// TIA Portal project "babu_mathQuestions" (V15)

(* hardware
DEVICE "S7-1200 station_1"  S7-1200 Station
   slot 0: "Rack_0"  S7-1200 Rack  Rack  V1.0
   slot 1: "PLC_1"  CPU 1212C DC/DC/DC  6ES7 212-1AE40-0XB0  V4.2
*)

// ===== PLC "PLC_1"  CPU 1212C DC/DC/DC =====

VAR_GLOBAL   // PLC tag table "Default tag table"
   "VAR1" AT %IW0 : Int;
   "INITIALIZE MEM" AT %M0.0 : Bool;
   "VAR21" AT %MW2 : Int;
   "VAR22" AT %MW4 : Int;
   "VAR23" AT %MW6 : Int;
   "VAR24" AT %MW8 : Int;
   "VAR31" AT %MD10 : Real;
   "VAR32" AT %MD14 : Real;
   "VAR33" AT %MD18 : Real;
   "VAR41" AT %MW22 : Int;
   "VAR42" AT %MW24 : Int;
   "VAR43" AT %MW26 : Int;
   "VAR44" AT %MW28 : Int;
   "VAR45" AT %MW30 : Int;
END_VAR

ORGANIZATION_BLOCK "Main"   // OB1, LAD, ProgramCycle
TITLE = "Main Program Sweep (Cycle)"
{ S7_Optimized_Access := 'TRUE' }
VERSION : 0.1
   VAR_INPUT
      Initial_Call : Bool;   // Initial call of this OB
      Remanence : Bool;   // =True, if remanent data are available
   END_VAR
BEGIN

REGION Network 1: INITIALIZE
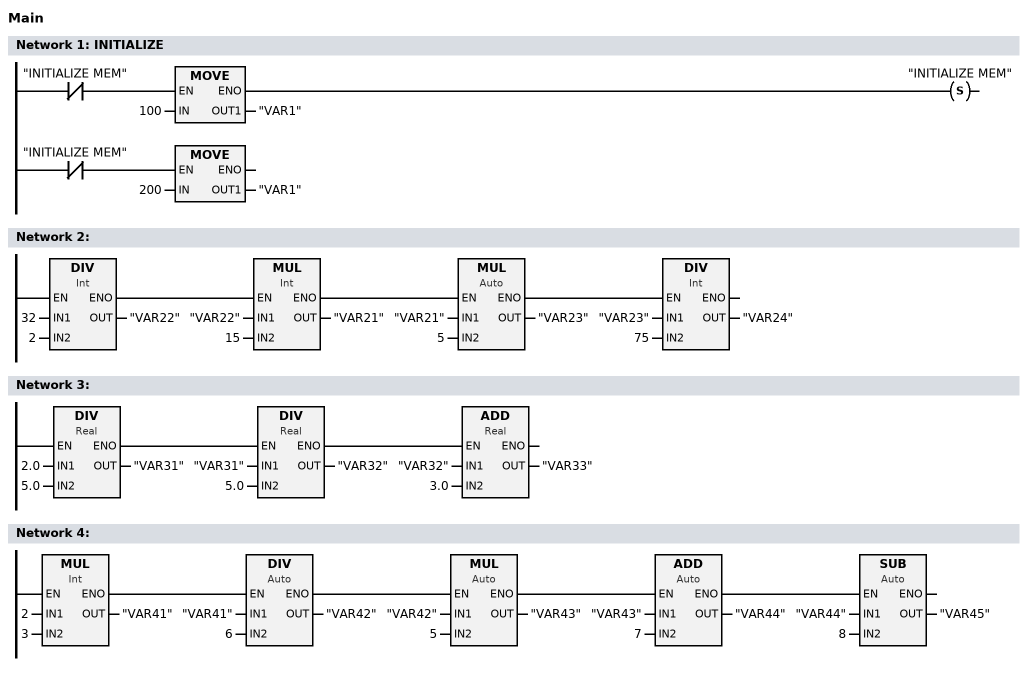
   RUNG wire#powerrail
      I_Contact( "INITIALIZE MEM" )
      Move(in := 100, out1 => "VAR1")
      S_Coil( "INITIALIZE MEM" )
   END_RUNG
   RUNG wire#powerrail
      I_Contact( "INITIALIZE MEM" )
      Move(in := 200, out1 => "VAR1")
   END_RUNG
   // the same network as SCL:
   IF NOT "INITIALIZE MEM" THEN
       "VAR1" := 100;
       "INITIALIZE MEM" := TRUE;
   END_IF;
   IF NOT "INITIALIZE MEM" THEN "VAR1" := 200; END_IF;
END_REGION

REGION Network 2
   RUNG wire#powerrail
      { S7_Templates := "SrcType := Int" } Div(in1 := 32, in2 := 2, out => "VAR22")
      { S7_Templates := "SrcType := Int" } Mul(in1 := "VAR22", in2 := 15, out => "VAR21")
      Mul(in1 := "VAR21", in2 := 5, out => "VAR23")
      { S7_Templates := "SrcType := Int" } Div(in1 := "VAR23", in2 := 75, out => "VAR24")
   END_RUNG
   // the same network as SCL:
   "VAR22" := 32 / 2;
   "VAR21" := "VAR22" * 15;
   "VAR23" := "VAR21" * 5;
   "VAR24" := "VAR23" / 75;
END_REGION

REGION Network 3
   RUNG wire#powerrail
      { S7_Templates := "SrcType := Real" } Div(in1 := 2.0, in2 := 5.0, out => "VAR31")
      { S7_Templates := "SrcType := Real" } Div(in1 := "VAR31", in2 := 5.0, out => "VAR32")
      { S7_Templates := "SrcType := Real" } Add(in1 := "VAR32", in2 := 3.0, out => "VAR33")
   END_RUNG
   // the same network as SCL:
   "VAR31" := 2.0 / 5.0;
   "VAR32" := "VAR31" / 5.0;
   "VAR33" := "VAR32" + 3.0;
END_REGION

REGION Network 4
   RUNG wire#powerrail
      { S7_Templates := "SrcType := Int" } Mul(in1 := 2, in2 := 3, out => "VAR41")
      Div(in1 := "VAR41", in2 := 6, out => "VAR42")
      Mul(in1 := "VAR42", in2 := 5, out => "VAR43")
      Add(in1 := "VAR43", in2 := 7, out => "VAR44")
      Sub(in1 := "VAR44", in2 := 8, out => "VAR45")
   END_RUNG
   // the same network as SCL:
   "VAR41" := 2 * 3;
   "VAR42" := "VAR41" / 6;
   "VAR43" := "VAR42" * 5;
   "VAR44" := "VAR43" + 7;
   "VAR45" := "VAR44" - 8;
END_REGION
END_ORGANIZATION_BLOCK